// Mitsubishi GX Developer project: PLC_PD_Controller   PLC: FX3U

PROGRAM MAIN
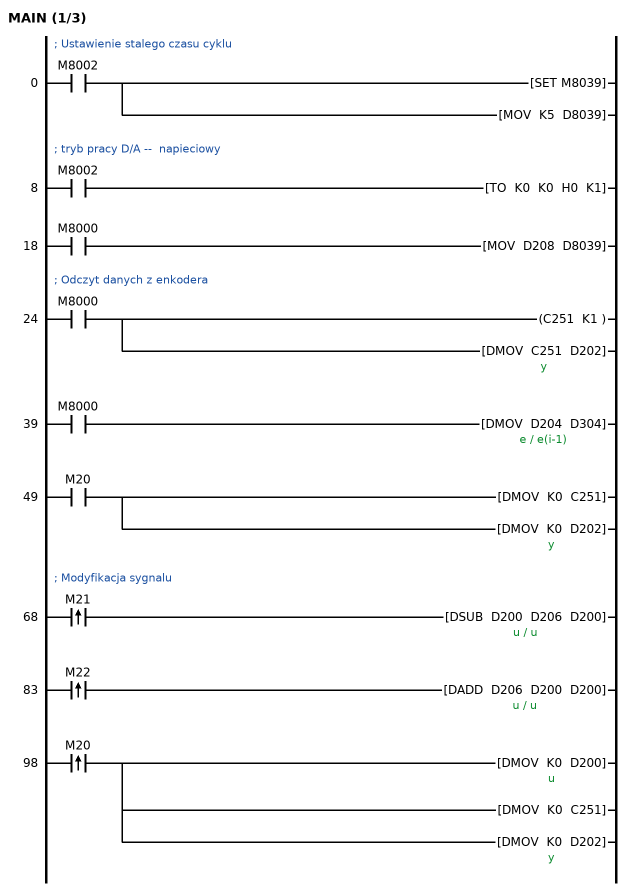
; Ustawienie stalego czasu cyklu
0     LD      M8002
      SET     M8039
      MOV     K5 D8039
; tryb pracy D/A --  napieciowy
8     LD      M8002
      TO      K0 K0 H0 K1
18    LD      M8000
      MOV     D208 D8039
; Odczyt danych z enkodera
24    LD      M8000
      OUT     C251 K1
      DMOV    C251 D202  ; y
39    LD      M8000
      DMOV    D204 D304  ; e / e(i-1)
49    LD      M20
      DMOV    K0 C251
      DMOV    K0 D202
; Modyfikacja sygnalu
68    LDP     M21
      DSUB    D200 D206 D200  ; u
83    LDP     M22
      DADD    D206 D200 D200
98    LDP     M20
      DMOV    K0 D200
      DMOV    K0 C251
      DMOV    K0 D202
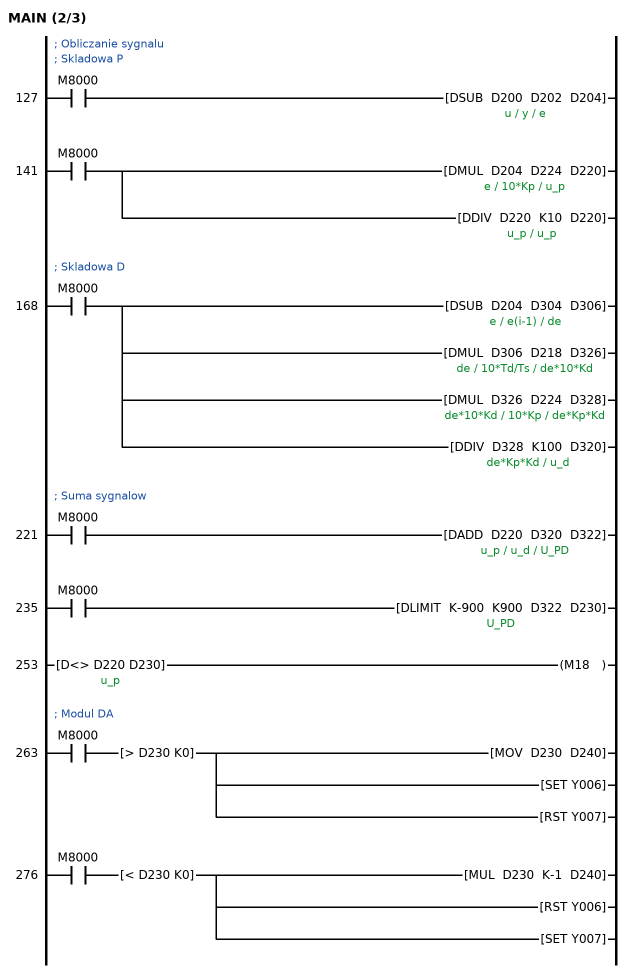
; Obliczanie sygnalu
; Skladowa P
127   LD      M8000
      DSUB    D200 D202 D204
141   LD      M8000
      DMUL    D204 D224 D220  ; 10*Kp / u_p
      DDIV    D220 K10 D220
; Skladowa D
168   LD      M8000
      DSUB    D204 D304 D306  ; de
      DMUL    D306 D218 D326  ; 10*Td/Ts / de*10*Kd
      DMUL    D326 D224 D328  ; de*Kp*Kd
      DDIV    D328 K100 D320  ; u_d
; Suma sygnalow
221   LD      M8000
      DADD    D220 D320 D322  ; U_PD
235   LD      M8000
      DLIMIT  K-900 K900 D322 D230
253   LDD<>   D220 D230  ; u_p
      OUT     M18
; Modul DA
263   LD      M8000
      AND>    D230 K0
      MOV     D230 D240
      SET     Y006
      RST     Y007
276   LD      M8000
      AND<    D230 K0
      MUL     D230 K-1 D240
      RST     Y006
      SET     Y007
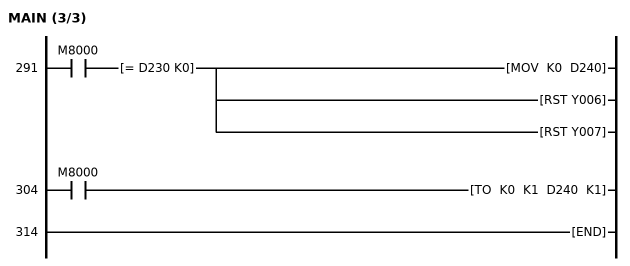
291   LD      M8000
      AND=    D230 K0
      MOV     K0 D240
      RST     Y006
      RST     Y007
304   LD      M8000
      TO      K0 K1 D240 K1
314   END
END_PROGRAM

// device comments not shown above
D214  ; Kp
D222  ; 10*Td/Ts
D324  ; 10*Td/Ts
